FUNCTION_BLOCK hysterisis
VAR_INPUT
	IN		: INT;
	thresh	: INT;
	variatie: INT;
END_VAR
VAR_OUTPUT
	UP		: BOOL;
END_VAR
VAR
END_VAR

IF IN > (thresh + variatie) THEN
	UP := TRUE;
ELSIF IN < (thresh - variatie) THEN
	UP := FALSE;
END_IF

END_FUNCTION_BLOCK

(* stored: Version 1.1.0.1, ProductVersion 3.1.4022.12
   POU hysterisis: Id {365db65f-c3c8-4fd0-8d42-5269775de037}, SpecialFunc None *)
